RoboDK station: cylinder_surface_test2.rdk

Station cylinder_surface_test2 (saved by RoboDK 5.0.0). Poses are relative to the parent item; angles as X-Y-Z fixed-axis rotations.
  - frame base frame at (230.5, -268.4, 259.1) mm, rotated rx -37.34 ry 33.83 rz -23.01 deg
  - frame p1 at (434.64, -113.95, 360.15) mm, rotated rx -37.34 ry 33.83 rz -23.01 deg
  - frame p2 at (726.57, -1.83, 967.9) mm, rotated rx -37.34 ry 33.83 rz -23.01 deg
  - frame out frame at (434.6, -113.9, 360.1) mm, rotated rx -12.3 ry -24.5 rz -131.3 deg
    - frame Frame 5 at (0, 0, 683.5) mm
